TYPE DUT_TASKSTATE :
(
	Unassigned := 0,
	//Assigned := 1,
	WaitingForSkillReady := 1,
	InProgress := 2,
	Done := 3,
	Aborted := 4,
	Error := 5
);
END_TYPE

(* stored: Version 1.1.0.1, ProductVersion 3.1.0.25
   DUT DUT_TASKSTATE: Id {e714243f-6753-4a1c-ad39-101cf979a80a} *)
